PROGRAM MAIN
VAR
END_VAR

END_PROGRAM

(* stored: Version 1.1.0.1
   POU MAIN: Id {cea8d541-7774-46a1-97b3-46a766d9ec0d} *)
